// TIA Portal V19 program export: 2 tag tables, 0 data types, 1 data blocks, 2 code blocks (in call order from the OBs), 4 instance data blocks

VAR_GLOBAL   // PLC tag table "Default tag table"
   Tag_1 AT %T1 : Timer;
END_VAR

VAR_GLOBAL   // PLC tag table "faceplate"
   "Start Button 0" AT %I0.0 : Bool;
   "Stop Button 0" AT %I0.1 : Bool;
   "Start Button 1" AT %I0.2 : Bool;
   "Stop Button 1" AT %I0.3 : Bool;
   "Start Button 2" AT %I0.4 : Bool;
   "Stop Button 2" AT %I0.5 : Bool;
   "Start Button 3" AT %I0.6 : Bool;
   "Stop Button 3" AT %I0.7 : Bool;
   "Belt Conveyor (4m) 0 (+)" AT %Q0.0 : Bool;
   "Belt Conveyor (4m) 0 (-)" AT %Q0.1 : Bool;
   "Belt Conveyor (4m) 1 (+)" AT %Q0.2 : Bool;
   "Belt Conveyor (4m) 1 (-)" AT %Q0.3 : Bool;
   "Belt Conveyor (4m) 2 (+)" AT %Q0.4 : Bool;
   "Belt Conveyor (4m) 2 (-)" AT %Q0.5 : Bool;
   "Belt Conveyor (4m) 3 (+)" AT %Q0.6 : Bool;
   "Belt Conveyor (4m) 3 (-)" AT %Q0.7 : Bool;
END_VAR

DATA_BLOCK "Controler Time"   // DB1
{ S7_Optimized_Access := 'TRUE' }
// stored: MemoryReserve 100
   VAR
      "Time-Right-Rest-con1" : Time := T#2s;
      "Time-Right-con1" : Time := T#3s;
      "Time-Left-con1" : Time := T#3s;
      "Time-Left-Rest-con1" : Time := T#2s;
      "Time-Right-con2" : Time := T#3s;
      "Time-Right-Rest-con2" : Time := T#2s;
      "Time-Left-con2" : Time := T#3s;
      "Time-Left-Rest-con2" : Time := T#2s;
      "Time-Right-con3" : Time := T#3s;
      "Time-Right-Rest-con3" : Time := T#2s;
      "Time-Left-con3" : Time := T#3s;
      "Time-Left-Rest-con3" : Time := T#2s;
      "Time-Right-con4" : Time := T#3s;
      "Time-Right-Rest-con4" : Time := T#2s;
      "Time-Left-con4" : Time := T#3s;
      "Time-Left-Rest-con4" : Time := T#2s;
      "mem-strat_1" : Bool;
      "mem-strat_2" : Bool;
      "mem-strat_3" : Bool;
      "mem-strat_4" : Bool;
      "mem-stop_1" : Bool;
      "mem-stop_2" : Bool;
      "mem-stop_3" : Bool;
      "mem-stop_4" : Bool;
   END_VAR
BEGIN
END_DATA_BLOCK

ORGANIZATION_BLOCK "Main"   // OB1, LAD, ProgramCycle
TITLE = "Main Program Sweep (Cycle)"
{ S7_Optimized_Access := 'TRUE' }
// stored: SetENOAutomatically false
   VAR_INPUT
      Initial_Call : Bool;   // Initial call of this OB
      Remanence : Bool;   // =True, if remanent data are available
   END_VAR
BEGIN

REGION Network 1
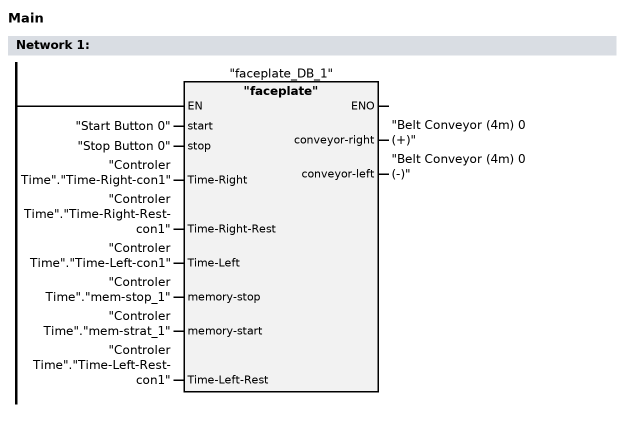
   RUNG wire#powerrail
      "faceplate_DB_1"(start := "Start Button 0", stop := "Stop Button 0", "Time-Right" := "Controler Time"."Time-Right-con1", "Time-Right-Rest" := "Controler Time"."Time-Right-Rest-con1", "Time-Left" := "Controler Time"."Time-Left-con1", "memory-stop" := "Controler Time"."mem-stop_1", "memory-start" := "Controler Time"."mem-strat_1", "Time-Left-Rest" := "Controler Time"."Time-Left-Rest-con1", "conveyor-right" => "Belt Conveyor (4m) 0 (+)", "conveyor-left" => "Belt Conveyor (4m) 0 (-)")
   END_RUNG
   // the same network as SCL:
   "faceplate_DB_1"(start := "Start Button 0",   // "faceplate"
                    stop := "Stop Button 0",
                    "Time-Right" := "Controler Time"."Time-Right-con1",
                    "Time-Right-Rest" := "Controler Time"."Time-Right-Rest-con1",
                    "Time-Left" := "Controler Time"."Time-Left-con1",
                    "memory-stop" := "Controler Time"."mem-stop_1",
                    "memory-start" := "Controler Time"."mem-strat_1",
                    "Time-Left-Rest" := "Controler Time"."Time-Left-Rest-con1",
                    "conveyor-right" => "Belt Conveyor (4m) 0 (+)",
                    "conveyor-left" => "Belt Conveyor (4m) 0 (-)");
END_REGION
END_ORGANIZATION_BLOCK

FUNCTION_BLOCK "faceplate"   // FB1, LAD
{ S7_Optimized_Access := 'TRUE' }
// stored: MemoryReserve 100, SetENOAutomatically false
   VAR_INPUT
      start : Bool;
      stop : Bool;
   END_VAR
   VAR_OUTPUT
      "conveyor-right" : Bool;
      "conveyor-left" : Bool;
   END_VAR
   VAR_IN_OUT
      "Time-Right" : Time;
      "Time-Right-Rest" : Time;
      "Time-Left" : Time;
      "memory-stop" : Bool;
      "memory-start" : Bool;
      "Time-Left-Rest" : Time;
   END_VAR
   VAR
      "Timer-Right" : TP_TIME;
      "Timer-Right-Rest" : TP_TIME;
      "Timer-Left" : TP_TIME;
      "Timer-Left-Rest" : TP_TIME;
      "mem-start" : Bool;
      "mem-stop" : Bool;
      "mem-edge-1" : Bool;
      "mem-edge-2" : Bool;
      "mem-edge-3" : Bool;
      "mem-edge-4" : Bool;
      "mem-edge-5" : Bool;
      "mem-edge-6" : Bool;
   END_VAR
   VAR_TEMP   // added for the SCL form of the ladder/FBD networks
      _w1 : Bool;
   END_VAR
BEGIN

REGION Network 1
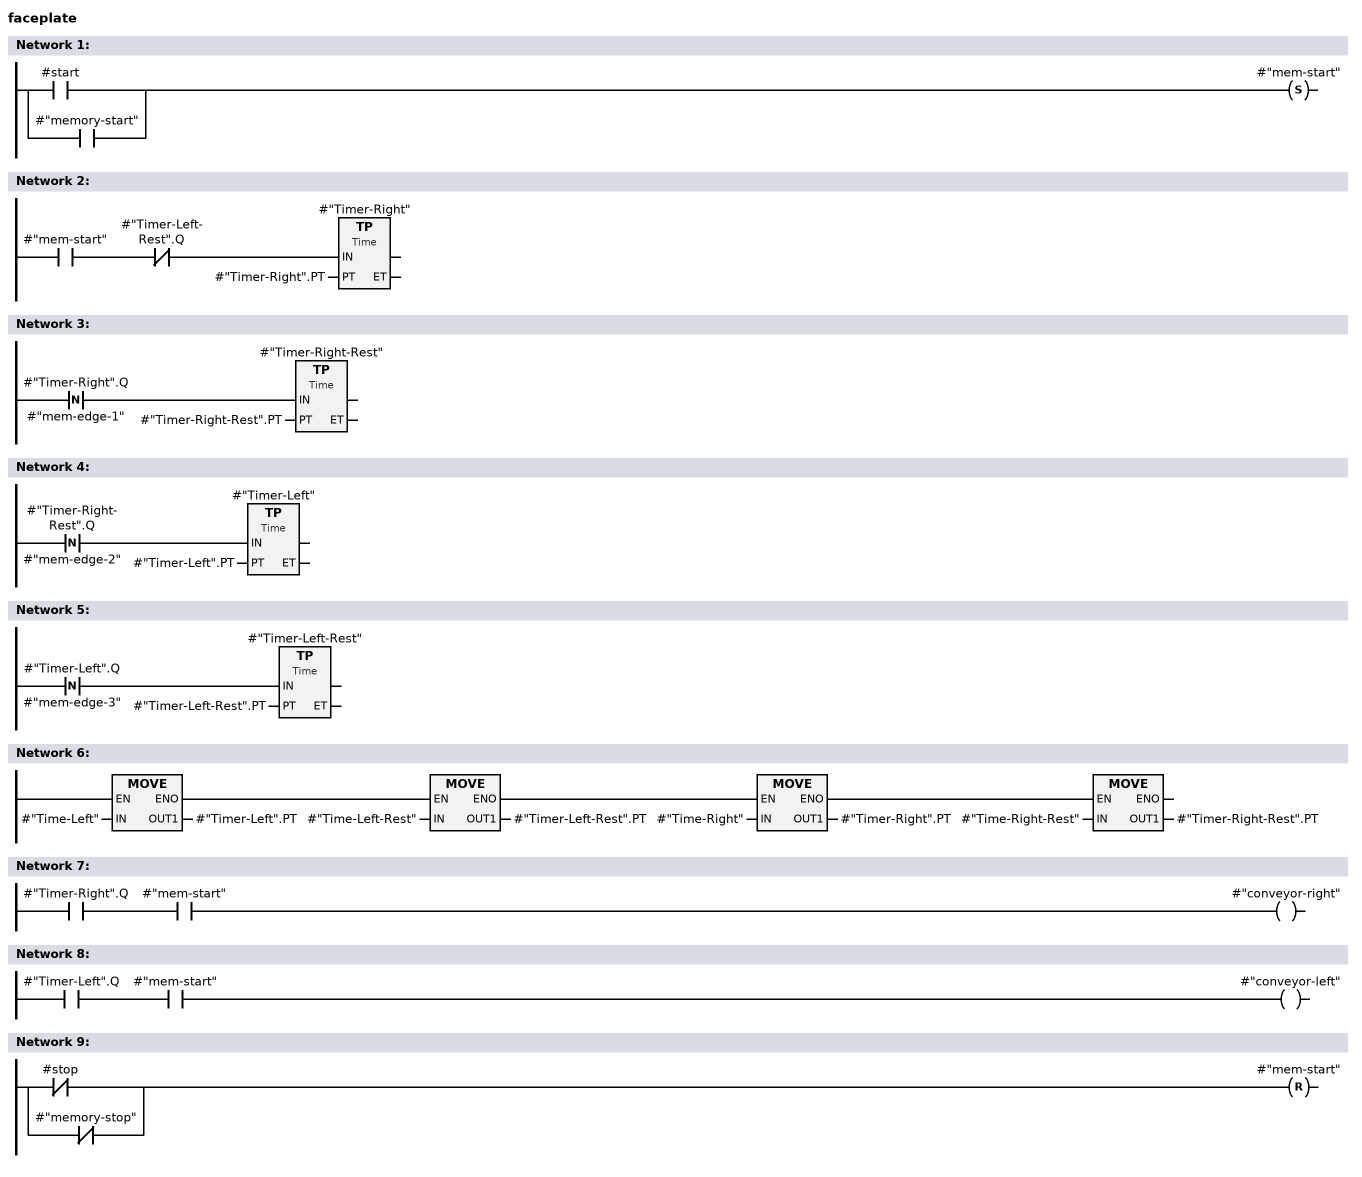
   RUNG wire#powerrail
      Contact( #start )
      wire#w1
      S_Coil( #"mem-start" )
   END_RUNG
   RUNG wire#powerrail
      Contact( #"memory-start" )
   END_RUNG wire#w1
   // the same network as SCL:
   IF #start OR #"memory-start" THEN #"mem-start" := TRUE; END_IF;
END_REGION

REGION Network 2
   RUNG wire#powerrail
      Contact( #"mem-start" )
      I_Contact( #"Timer-Left-Rest".Q )
      { S7_Templates := "time_type := Time" } #"Timer-Right".TP(pt := #"Timer-Right".PT, et =>)
   END_RUNG
   // the same network as SCL:
   #"Timer-Right"(IN := #"mem-start" AND NOT #"Timer-Left-Rest".Q, PT := #"Timer-Right".PT);   // TP
END_REGION

REGION Network 3
   RUNG wire#powerrail
      N_Contact(operand := #"Timer-Right".Q, bit := #"mem-edge-1")
      { S7_Templates := "time_type := Time" } #"Timer-Right-Rest".TP(pt := #"Timer-Right-Rest".PT, et =>)
   END_RUNG
   // the same network as SCL:
   #_w1 := NOT #"Timer-Right".Q AND #"mem-edge-1";   // falling edge of #"Timer-Right".Q
   #"mem-edge-1" := #"Timer-Right".Q;
   #"Timer-Right-Rest"(IN := #_w1, PT := #"Timer-Right-Rest".PT);   // TP
END_REGION

REGION Network 4
   RUNG wire#powerrail
      N_Contact(operand := #"Timer-Right-Rest".Q, bit := #"mem-edge-2")
      { S7_Templates := "time_type := Time" } #"Timer-Left".TP(pt := #"Timer-Left".PT, et =>)
   END_RUNG
   // the same network as SCL:
   #_w1 := NOT #"Timer-Right-Rest".Q AND #"mem-edge-2";   // falling edge of #"Timer-Right-Rest".Q
   #"mem-edge-2" := #"Timer-Right-Rest".Q;
   #"Timer-Left"(IN := #_w1, PT := #"Timer-Left".PT);   // TP
END_REGION

REGION Network 5
   RUNG wire#powerrail
      N_Contact(operand := #"Timer-Left".Q, bit := #"mem-edge-3")
      { S7_Templates := "time_type := Time" } #"Timer-Left-Rest".TP(pt := #"Timer-Left-Rest".PT, et =>)
   END_RUNG
   // the same network as SCL:
   #_w1 := NOT #"Timer-Left".Q AND #"mem-edge-3";   // falling edge of #"Timer-Left".Q
   #"mem-edge-3" := #"Timer-Left".Q;
   #"Timer-Left-Rest"(IN := #_w1, PT := #"Timer-Left-Rest".PT);   // TP
END_REGION

REGION Network 6
   RUNG wire#powerrail
      Move(in := #"Time-Left", out1 => #"Timer-Left".PT)
      Move(in := #"Time-Left-Rest", out1 => #"Timer-Left-Rest".PT)
      Move(in := #"Time-Right", out1 => #"Timer-Right".PT)
      Move(in := #"Time-Right-Rest", out1 => #"Timer-Right-Rest".PT)
   END_RUNG
   // the same network as SCL:
   #"Timer-Left".PT := #"Time-Left";
   #"Timer-Left-Rest".PT := #"Time-Left-Rest";
   #"Timer-Right".PT := #"Time-Right";
   #"Timer-Right-Rest".PT := #"Time-Right-Rest";
END_REGION

REGION Network 7
   RUNG wire#powerrail
      Contact( #"Timer-Right".Q )
      Contact( #"mem-start" )
      Coil( #"conveyor-right" )
   END_RUNG
   // the same network as SCL:
   #"conveyor-right" := #"Timer-Right".Q AND #"mem-start";
END_REGION

REGION Network 8
   RUNG wire#powerrail
      Contact( #"Timer-Left".Q )
      Contact( #"mem-start" )
      Coil( #"conveyor-left" )
   END_RUNG
   // the same network as SCL:
   #"conveyor-left" := #"Timer-Left".Q AND #"mem-start";
END_REGION

REGION Network 9
   RUNG wire#powerrail
      I_Contact( #stop )
      wire#w1
      R_Coil( #"mem-start" )
   END_RUNG
   RUNG wire#powerrail
      I_Contact( #"memory-stop" )
   END_RUNG wire#w1
   // the same network as SCL:
   IF NOT #stop OR NOT #"memory-stop" THEN #"mem-start" := FALSE; END_IF;
END_REGION
END_FUNCTION_BLOCK

DATA_BLOCK "faceplate_DB"   // DB2
// stored: InstanceOfName faceplate, InstanceOfType FB
"faceplate"
BEGIN
END_DATA_BLOCK

DATA_BLOCK "faceplate_DB_1"   // DB3
// stored: InstanceOfName faceplate, InstanceOfType FB
"faceplate"
BEGIN
END_DATA_BLOCK

DATA_BLOCK "faceplate_DB_2"   // DB4
// stored: InstanceOfName faceplate, InstanceOfType FB
"faceplate"
BEGIN
END_DATA_BLOCK

DATA_BLOCK "faceplate_DB_3"   // DB5
// stored: InstanceOfName faceplate, InstanceOfType FB
"faceplate"
BEGIN
END_DATA_BLOCK
